Staubli VAL3: CUTIN.pgx

public program CutIn(trsf x_trCenter, trsf& x_trLine[], trsf& x_trDest[], trsf& x_trCut, num x_nType, num x_nPercent, bool& x_bRes)
  local pointRx l_trCutInP
  local frame l_fFrame
  local trsf l_trBuff[3]
  local num l_nR
begin
  //切入引线
  //x_nType==0  无引线
  //==1   直线
  //==2   圆弧


  //如果是直线，直接退出
  if x_nType==0
    x_bRes=true
    return
  else
    x_bRes=false
  endIf


  //参数合法性判断
  if x_nType<0 or x_nType>2
    return
  endIf



  //根据三点求用户坐标系
  l_trBuff[0]=x_trLine[0]
  l_trBuff[1]=x_trLine[1]
  l_trBuff[2]=x_trCenter

  call SetFrame(l_trBuff,l_fFrame,x_bRes)
  if !x_bRes
    return
  endIf

  //**********************************
  //2014.10.23
  //从圆心开始调整
  //为切厚板改写的程序
  if  x_nPercent==101
    //2015.01.22
    //添加新的变量来支持厚板切割
    //厚板切割内切圆的圆心的长度
    if distance(x_trLine[0],x_trCenter)<=max(5,nThickRadio)
      x_trDest[0]=x_trCenter
    else
      l_trCutInP.trsf={0,10,0,0,0,0}
      link(l_trCutInP,l_fFrame)
      x_trDest[0]=position(l_trCutInP,world)
    endIf
    return
  endIf

  //*********************************





  l_trCutInP.trsf=x_trCenter
  link(l_trCutInP,world)
  l_trCutInP.trsf=position(l_trCutInP,l_fFrame)
  //2014.7.24
  l_nR=min(abs(l_trCutInP.trsf.y)/2,10)
  //l_nR=min(abs(l_trCutInP.trsf.y),10)


  if l_nR==0
    x_bRes=false
    return
  endIf

  //切入切出比例
  if x_nPercent>0 and x_nPercent<100

    l_nR=l_nR*x_nPercent/100
  endIf


  l_trCutInP.trsf.y=0
  link(l_trCutInP,l_fFrame)
  l_trCutInP.trsf=position(l_trCutInP,world)

  x_trCut=l_trCutInP.trsf


  l_trBuff[0]=l_trCutInP.trsf
  call SetFrame(l_trBuff,l_fFrame,x_bRes)
  if !x_bRes
    return
  endIf

  l_trCutInP.trsf={-l_nR,l_nR,0,0,0,0}
  link(l_trCutInP,l_fFrame)
  x_trDest[0]=position(l_trCutInP,world)

  if x_nType==2
    l_trCutInP.trsf={-sin(45)*l_nR,l_nR-sin(45)*l_nR,0,0,0,0}
    link(l_trCutInP,l_fFrame)
    x_trDest[1]=position(l_trCutInP,world)
  endIf

end
